FUNCTION_BLOCK differential_protection_1_4 (* Composite Function Block Type *)
  (* Standard: 61499-2 *)
  (* Version 0.0, 3/23/2016, gulzha, nxtControl GmbH, template *)
  PACKAGE Main;
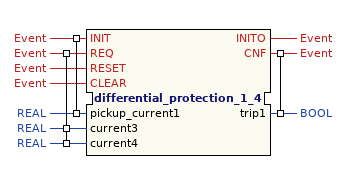
  EVENT_INPUT
    INIT WITH pickup_current1; (* Initialization Request *)
    REQ WITH current3, current4; (* Normal Execution Request *)
    RESET;
    CLEAR;
  END_EVENT
  EVENT_OUTPUT
    INITO; (* Initialization Confirm *)
    CNF WITH trip1; (* Execution Confirmation *)
  END_EVENT
  VAR_INPUT
    pickup_current1 : REAL;
    current3 : REAL;
    current4 : REAL;
  END_VAR
  VAR_OUTPUT
    trip1 : BOOL;
  END_VAR
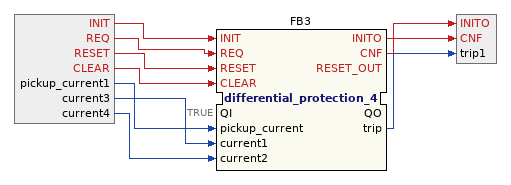
  FBS
    FB3 : differential_protection_4(QI := TRUE);
  END_FBS
  EVENT_CONNECTIONS
    FB3.INITO TO INITO;
    FB3.CNF TO CNF;
    INIT TO FB3.INIT;
    REQ TO FB3.REQ;
    RESET TO FB3.RESET;
    CLEAR TO FB3.CLEAR;
  END_CONNECTIONS
  DATA_CONNECTIONS
    FB3.trip TO trip1;
    pickup_current1 TO FB3.pickup_current;
    current3 TO FB3.current1;
    current4 TO FB3.current2;
  END_CONNECTIONS
END_FUNCTION_BLOCK
